TYPE T_Ctrl_SIf_PTS_Ilk :
STRUCT
END_STRUCT
END_TYPE

(* stored: Version 1.1.0.1, ProductVersion 3.1.0.25
   DUT T_Ctrl_SIf_PTS_Ilk: Id {2a38859f-d5f9-4289-98ef-01ec4024bce0} *)
